(* IEC 61131-3 sources: vscode-st/examples/15-multi-file, 4 files *)

(* ---- types.st ---- *)
/* 15-multi-file/types.st — Shared type declarations
   Types referenced across the multi-file project. */

TYPE MotorState : (Stopped, Starting, Running, Stopping, Error); END_TYPE

TYPE MotorConfig : STRUCT
    maxSpeed   : REAL    := 3000.0;
    accelRate  : REAL    := 5.0;
    decelRate  : REAL    := 10.0;
    state      : MotorState;
END_STRUCT; END_TYPE

(* ---- globals.st ---- *)
/* 15-multi-file/globals.st — Shared global declarations
   These GVLs are referenced by other files in this multi-file example. */

VAR_GLOBAL
    gSystemTick     : DINT;
    gEmergencyStop  : BOOL;
    gLineSpeed      : REAL  := 100.0;
END_VAR

VAR_GLOBAL CONSTANT
    gMaxConveyors   : INT   := 16;
    gWatchdogMs     : TIME  := T#200ms;
END_VAR

(* ---- motor_fb.st ---- *)
/* 15-multi-file/motor_fb.st — Function block referencing
   external globals and types from other files. Uses CASE
   for state-machine logic. */

FUNCTION_BLOCK MotorController
VAR_INPUT
    startCmd     : BOOL;
    stopCmd      : BOOL;
    speedRef     : REAL;
END_VAR
VAR_OUTPUT
    running      : BOOL;
    actualSpeed  : REAL;
    fault        : BOOL;
END_VAR
VAR
    config       : MotorConfig;    // From types.st
    rampStep     : REAL;
END_VAR

// Reference global from globals.st
IF gEmergencyStop THEN
    running := FALSE;
    actualSpeed := 0.0;
    fault := TRUE;
    RETURN;
END_IF;

// State machine using CASE
CASE config.state OF
    MotorState.Stopped:
        IF startCmd AND NOT stopCmd THEN
            config.state := MotorState.Starting;
            running := TRUE;
        END_IF;

    MotorState.Starting:
        actualSpeed := actualSpeed + config.accelRate * 0.01;
        IF actualSpeed >= speedRef THEN
            actualSpeed := speedRef;
            config.state := MotorState.Running;
        END_IF;

    MotorState.Running:
        IF stopCmd THEN
            config.state := MotorState.Stopping;
        END_IF;

    MotorState.Stopping:
        actualSpeed := actualSpeed - config.decelRate * 0.01;
        IF actualSpeed <= 0.0 THEN
            actualSpeed := 0.0;
            config.state := MotorState.Stopped;
            running := FALSE;
        END_IF;

    MotorState.Error:
        running := FALSE;
        actualSpeed := 0.0;
END_CASE;

END_FUNCTION_BLOCK

(* ---- line_control.st ---- *)
/* 15-multi-file/line_control.st — Main PROGRAM
   References globals, types, and FBs from other files
   in the multi-file project. */

PROGRAM LineControl
VAR
    motor1      : MotorController;   // From motor_fb.st
    motor2      : MotorController;   // From motor_fb.st
    lineRunning : BOOL;
    startBtn    AT %IX0.0 : BOOL;
    stopBtn     AT %IX0.1 : BOOL;
    speedPot    AT %IW2   : INT;
    reqSpeed    : REAL;
END_VAR

// Convert analog input to speed reference
reqSpeed := INT_TO_REAL(speedPot) * (gLineSpeed / REAL#100.0);

// Control motor 1
motor1(
    startCmd := startBtn AND NOT stopBtn AND NOT gEmergencyStop,
    stopCmd  := stopBtn OR gEmergencyStop,
    speedRef := reqSpeed
);

// Control motor 2 with offset
motor2(
    startCmd := startBtn AND NOT stopBtn AND NOT gEmergencyStop
                AND motor1.running,
    stopCmd  := stopBtn OR gEmergencyStop
                OR motor1.fault,
    speedRef := reqSpeed * REAL#0.95
);

lineRunning := motor1.running AND motor2.running;

// System monitoring using globals
gSystemTick := gSystemTick + 1;

END_PROGRAM
